// TwinCAT 3 PLC project AbstractObjectTestLib
// Title: AbstractObjectTestLib
// Company: ekvip automation GmbH
// Author: tdie
// ProjectVersion: 4.0.0.0
// Description: UnitTest library for basic IObject-Interface tests .. <legal notes> legal notes ================= | SPDX-FileCopyrightText: © 2022 ekvip automation GmbH <info@ekvip.de> | SPDX-License-Identifier: Apache-2.0 | For details check: Apache-2.0_ .. _Apache-2.0: https://www.apache.org/licenses/LICENSE-2.0 .. </legal notes>
// ProgramVersion: 3.1.4026.11
// libraries:
//   CNM_AbstractObject, * (ekvip automation GmbH)
//   CNM_ReturnTypes, * (ekvip automation GmbH)
//   Tc2_Standard, * (Beckhoff Automation GmbH)
//   Tc2_System, * (Beckhoff Automation GmbH)
//   Tc2_Utilities, * (Beckhoff Automation GmbH)
//   TcUnit, * (www.tcunit.org)
// project tree:
//   StupidObject/classes/ StupidObject.TcPOU (not stored)
//   StupidObject/interfaces/ IStupidObject1.TcIO, IStupidObject2.TcIO, IStupidObject3.TcIO, IStupidObject4.TcIO (not stored)
//   Tests/ AbstractObject_Test.TcPOU (not stored)

// ---- StupidObject/interfaces/IStupidObject1.TcIO
(*

short summary
=================
This is a useless interface for the validity test.

.. <legal notes>

legal notes
=================
| SPDX-FileCopyrightText: © 2024 ekvip automation GmbH <info@ekvip.de>
| SPDX-License-Identifier: Apache-2.0
| For details check: Apache-2.0_

.. _Apache-2.0: https://www.apache.org/licenses/LICENSE-2.0

.. </legal notes>

*)

INTERFACE INTERNAL IStupidObject1 EXTENDS CNM_AbstractObject.IObject

END_INTERFACE

// ---- StupidObject/interfaces/IStupidObject2.TcIO
(*

short summary
=================
This is a useless interface for the validity test.

.. <legal notes>

legal notes
=================
| SPDX-FileCopyrightText: © 2024 ekvip automation GmbH <info@ekvip.de>
| SPDX-License-Identifier: Apache-2.0
| For details check: Apache-2.0_

.. _Apache-2.0: https://www.apache.org/licenses/LICENSE-2.0

.. </legal notes>

*)

INTERFACE INTERNAL IStupidObject2 EXTENDS CNM_AbstractObject.IObject

END_INTERFACE

// ---- StupidObject/interfaces/IStupidObject3.TcIO
(*

short summary
=================
This is a useless interface for the validity test.

.. <legal notes>

legal notes
=================
| SPDX-FileCopyrightText: © 2024 ekvip automation GmbH <info@ekvip.de>
| SPDX-License-Identifier: Apache-2.0
| For details check: Apache-2.0_

.. _Apache-2.0: https://www.apache.org/licenses/LICENSE-2.0

.. </legal notes>

*)

INTERFACE INTERNAL IStupidObject3 EXTENDS CNM_AbstractObject.IObject

END_INTERFACE
